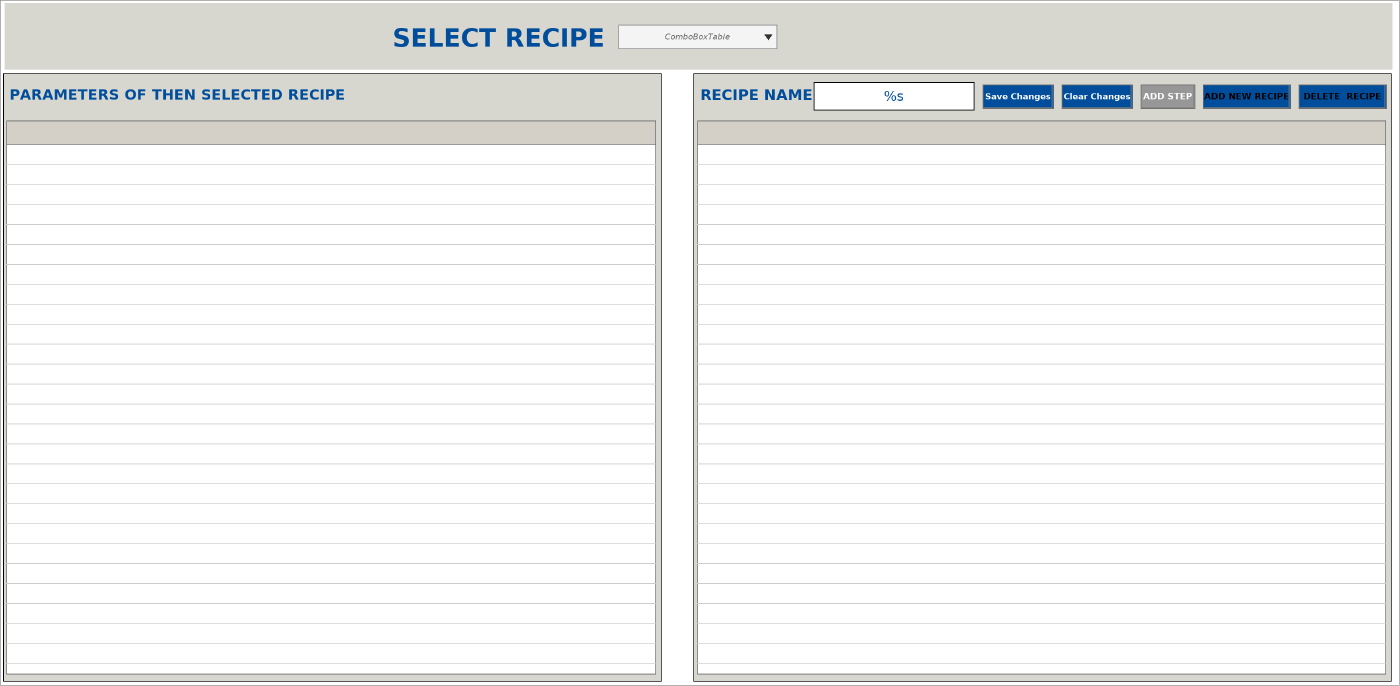
VISUALIZATION Recipe  // 1755x860
    RoundedRectangle (6,4 1739x83)
    Rectangle (491,22 268x51), "SELECT RECIPE"
    Rectangle (4,92 825x762)
    Table (8,151 814x694), data array: gRecipeViewData
        p1128707560: gShowNum
        p3854506369: gRecipeViewData[INDEX].NUM
        p1892666644: gRecipeViewData[INDEX].etchTime
        p338671338: gRecipeViewData[INDEX].rfPoint_Source
        p2170511999: gRecipeViewData[INDEX].pdvPoint
        p3723444502: gRecipeViewData[INDEX].mfc1
        p1218418051: gRecipeViewData[INDEX].mfc2
        p746581629: gRecipeViewData[INDEX].mfc3
        p3104783080: gRecipeViewData[INDEX].mfc4
        p2501879983: gRecipeViewData[INDEX].mfc5
        p7306298: gRecipeViewData[INDEX].mfc6
        p1933151965: gRecipeViewData[INDEX].mfc7
        p3863566920: gRecipeViewData[INDEX].mfc8
        p2192122294: gRecipeViewData[INDEX].mfc9
        p400160035: gRecipeViewData[INDEX].rfPoint_Power
        p1265227338: gRecipeViewData[INDEX].par_2
        p3726181087: gRecipeViewData[INDEX].par_3
        p3136911649: gRecipeViewData[INDEX].par_4
        p2237128397: N2(50)
        p505689113: CF4(200)
        p1757482276: CHF3(200)
        p4088588272: SF6(200)
        p2243050616: O2(100)
        p516019884: O2(10)
        p1739542657: He(500)
        p4242324053: Ar(500)
        p2319025000: C4F8(200)
        p3312258591: gRecipeViewData[INDEX].par1
        p1791247317: gRecipeViewData[INDEX].par2
        p262371475: gRecipeViewData[INDEX].par3
        p4008173056: gRecipeViewData[INDEX].par4
        p2340480326: gRecipeViewData[INDEX].par5
        p606709900: gRecipeViewData[INDEX].par6
        p1095668682: gRecipeViewData[INDEX].par7
        p1037165547: gRecipeViewData[INDEX].par8
        p1488378029: gRecipeViewData[INDEX].par9
        p152217274: gRecipeViewData[INDEX].par10
        p1819647484: gRecipeViewData[INDEX].par11
        p3286028342: gRecipeViewData[INDEX].par12
        p2797333360: gRecipeViewData[INDEX].par13
        p1207913955: gRecipeViewData[INDEX].par14
        p580417189: gRecipeViewData[INDEX].par15
        p2368813935: gRecipeViewData[INDEX].par16
    Rectangle (9,99 424x40), "PARAMETERS OF THEN SELECTED RECIPE"
    Rectangle (869,92 875x762)
    Table (874,151 863x694), data array: gRecipeEditorData
        p1128707560: gShowNum
        p1420305297: gselectclo
        p1137915858: gselectRow
        p2664070770: Delete
        p3854506369: gRecipeEditorData[INDEX].NUM
        p1892666644: gRecipeEditorData[INDEX].etchTime
        p338671338: gRecipeEditorData[INDEX].rfPoint_Source
        p2170511999: gRecipeEditorData[INDEX].pdvPoint
        p3723444502: gRecipeEditorData[INDEX].mfc1
        p1218418051: gRecipeEditorData[INDEX].mfc2
        p746581629: gRecipeEditorData[INDEX].mfc3
        p3104783080: gRecipeEditorData[INDEX].mfc4
        p2501879983: gRecipeEditorData[INDEX].mfc5
        p7306298: gRecipeEditorData[INDEX].mfc6
        p1933151965: gRecipeEditorData[INDEX].mfc7
        p3863566920: gRecipeEditorData[INDEX].mfc8
        p2192122294: gRecipeEditorData[INDEX].mfc9
        p400160035: gRecipeEditorData[INDEX].rfPoint_Power
        p1265227338: gRecipeEditorData[INDEX].par_2
        p3726181087: gRecipeEditorData[INDEX].par_3
        p3136911649: gRecipeEditorData[INDEX].par_4
        p2237128397: N2(50)
        p505689113: CF4(200)
        p1757482276: CHF3(200)
        p4088588272: SF6(200)
        p2243050616: O2(100)
        p516019884: O2(10)
        p1739542657: He(500)
        p4242324053: Ar(500)
        p2319025000: C4F8(200)
        p3312258591: gRecipeEditorData[INDEX].par1
        p1791247317: gRecipeEditorData[INDEX].par2
        p262371475: gRecipeEditorData[INDEX].par3
        p4008173056: gRecipeEditorData[INDEX].par4
        p2340480326: gRecipeEditorData[INDEX].par5
        p606709900: gRecipeEditorData[INDEX].par6
        p1095668682: gRecipeEditorData[INDEX].par7
        p1037165547: gRecipeEditorData[INDEX].par8
        p1488378029: gRecipeEditorData[INDEX].par9
        p152217274: gRecipeEditorData[INDEX].par10
        p1819647484: gRecipeEditorData[INDEX].par11
        p3286028342: gRecipeEditorData[INDEX].par12
        p2797333360: gRecipeEditorData[INDEX].par13
        p1207913955: gRecipeEditorData[INDEX].par14
        p580417189: gRecipeEditorData[INDEX].par15
        p2368813935: gRecipeEditorData[INDEX].par16
        Columns.Column.[0].Template: OnMouseClick: write the text variable via Default
        Columns.Column.[1].Template: OnMouseClick: write the text variable via Default
        Columns.Column.[10].Template: OnMouseClick: write the text variable via Default
        Columns.Column.[11].Template: OnMouseClick: write the text variable via Default
        Columns.Column.[12].Template: OnMouseClick: write the text variable via Default
        Columns.Column.[13].Template: OnMouseClick: write the text variable via Default
        Columns.Column.[14].Template: OnMouseClick: write the text variable via Default
        Columns.Column.[15].Template: OnMouseClick: write the text variable via Default
        Columns.Column.[16].Template: OnMouseClick: execute { DataSave.fbDataSaveModule_EX_recipe.recipeStepDelete:=true; }
        Columns.Column.[2].Template: OnMouseClick: write the text variable via Default
        Columns.Column.[3].Template: OnMouseClick: write the text variable via Default
        Columns.Column.[4].Template: OnMouseClick: write the text variable via Default
        Columns.Column.[5].Template: OnMouseClick: write the text variable via Default
        Columns.Column.[6].Template: OnMouseClick: write the text variable via Default
        Columns.Column.[7].Template: OnMouseClick: write the text variable via Default
        Columns.Column.[8].Template: OnMouseClick: write the text variable via Default
        Columns.Column.[9].Template: OnMouseClick: write the text variable via Default
    Rectangle (875,99 143x40), "RECIPE NAME"
    RoundedRectangle (1020,103 201x35), "%s", text variable: gRecipeShowNameNow
        OnMouseClick: write the text variable via Default
    Button (1430,106 68x30), "ADD STEP"
        OnMouseClick: execute {
            gShowNum:=gShowNum+1;
            IF gShowNum>gRecipeStepMaxShow THEN
            	gShowNum:=gShowNum-1;
            	error_Trigger(1);
            ELSE
            	;
            END_IF
            DataSave.fbDataSaveModule_EX_recipe.addRecipeStep(gShowNum);
        }
    Button (1232,106 89x30), "Save Changes"
        OnMouseClick: execute { DataSave.fbDataSaveModule_EX_recipe.saveAct:=true; }
    Button (1331,106 89x30), "Clear Changes"
        OnMouseClick: execute {
            IF NOT DataSave.fbDataSaveModule_EX_recipename.busy THEN
            	DataSave.fbDataSaveModule_EX_recipename.readB:=true;
            END_IF
            IF NOT DataSave.fbDataSaveModule_EX_recipe.busy THEN
            	DataSave.fbDataSaveModule_EX_recipe.readB:=true;
            END_IF
        }
    Button (1508,106 110x30), "ADD NEW RECIPE"
        OnMouseClick: execute { DataSave.fbDataSaveModule_EX_recipe.addSlector(outrecipeSelect:=gRecipeNameSelect,outrecipeSelectShow:=gRecipeNameSelectShow,newName:=gRecipeShowNameNow); }
    Button (1628,106 110x30), "DELETE RECIPE"
        OnMouseClick: execute { DataSave.fbDataSaveModule_EX_recipe.deleteB:=TRUE; DataSave.fbDataSaveModule_EX_recipe.deleteSlector(recipeSelect:=gRecipeNameSelect,recipeSelectShow:=gRecipeNameSelectShow,inidex:=gRecipeSelectIndex1,outrecipeSelect=>gRecipeNameSelect,outrecipeSelectShow=>gRecipeNameSelectShow); }
    ComboBoxTable (775,31 199x30), variable: gRecipeSelectIndex1, data array: gRecipeNameSelect
        p1128707560: gRecipeSelctMaxIndex
        p3854506369: gRecipeNameSelect[INDEX].Name
END_VISUALIZATION

(* stored: Version 1.1.0.1, ProductVersion 3.1.4024.12
   Visu Recipe: Id {e6d7b0d9-c91b-4387-9ae1-373ccb8a1b40} *)
